// TIA Portal V16 export
// export: Created 2023-03-29T11:03:43.8543133Z, ExportSetting WithDefaults, DisplayName Totally Integrated Automation Portal, DisplayVersion V16 Update 6, DisplayName TIA Portal Version Control Interface, DisplayVersion V16 Update 2, DisplayName TIA Portal Openness, DisplayVersion V16 Update 6, DisplayName STEP 7 Professional, DisplayVersion V16 Update 6, DisplayName STEP 7 Safety, DisplayVersion V16, DisplayName WinCC Advanced, DisplayVersion V16 Update 6
VAR_GLOBAL   // PLC tag table "Default tag table"
   System_Byte AT %MB1 : Byte;
   FirstScan AT %M1.0 : Bool;
   DiagStatusUpdate AT %M1.1 : Bool;
   AlwaysTRUE AT %M1.2 : Bool;
   AlwaysFALSE AT %M1.3 : Bool;
   Clock_Byte AT %MB0 : Byte;
   Clock_10Hz AT %M0.0 : Bool;
   Clock_5Hz AT %M0.1 : Bool;
   "Clock_2.5Hz" AT %M0.2 : Bool;
   Clock_2Hz AT %M0.3 : Bool;
   "Clock_1.25Hz" AT %M0.4 : Bool;
   Clock_1Hz AT %M0.5 : Bool;
   "Clock_0.625Hz" AT %M0.6 : Bool;
   "Clock_0.5Hz" AT %M0.7 : Bool;
   trig_ustaw_czas AT %M206.1 : Bool;
   trig_pobierz_czas AT %M206.3 : Bool;
   "Bit_6-Wekt-Valve01_R" AT %M2000.6 : Bool;   // Bit-6 kasowanie alarmu
   "Bit_7-Wekt-Valve01_R" AT %M2000.7 : Bool;   // Bit trybu pracy napędu
   "Bit_5-Wekt-Valve01_R" AT %M2000.5 : Bool;   // Rozkaz zamykania
   "Bit_4-Wek_Valve01_R" AT %M2000.4 : Bool;   // Rozkaz otwieranie
   "Bit_0-Wekt_Valve01_R" AT %M2000.0 : Bool;   // Bit gotowośći / awarii
   "Bit_0-Wekt_Valve01_L" AT %M2001.0 : Bool;   // Bit Alarm/Gotowość (Alarm-=1, gotowość=0)
   "Bit_1-Wekt_Valve01_L" AT %M2001.1 : Bool;   // Bit potwierdzenia otwarcia
   "Bit_2-Wekt_Valve01_L" AT %M2001.2 : Bool;   // Bit wyboru trybu Zdalne=1 Remontowe=0
   "Bit_3-Wek_Valve01_L" AT %M2001.3 : Bool;   // Bit potwierdzenia zamknięcia
   "Bit_4-Wek_Valve01_L" AT %M2001.4 : Bool;   // Bit rozkazu na otwieranie
   "Bit_5-Wekt-Valve01_L" AT %M2001.5 : Bool;   // Bit rozkazu na zamykanie
   "Bit_6-Wekt-Valve01_L" AT %M2001.6 : Bool;   // Bit kasowania
   "Bit_7-Wekt-Valve01_L" AT %M2001.7 : Bool;   // Bit rodzaju sterowania aut =1 /manual= 0
   Byte_Wekt_Valve01_L AT %MB2001 : Byte;   // Lewy byte wektora napędu
   Byte_Wekt_Valve01_R AT %MB2000 : Byte;   // Prawy byte wektora napędu
   "I0.3" AT %I0.3 : Bool;
   "I0.4" AT %I0.4 : Bool;
   "I0.5" AT %I0.5 : Bool;
   "I0.6" AT %I0.6 : Bool;
   "Q0.3" AT %Q0.3 : Bool;
   "Q0.4" AT %Q0.4 : Bool;
   "Q0.5" AT %Q0.5 : Bool;
   "I6.4" AT %I6.4 : Bool;
   "I6.3" AT %I6.3 : Bool;
   "I6.2" AT %I6.2 : Bool;
   "I9.5" AT %I9.5 : Bool;
   "I9.6" AT %I9.6 : Bool;
   "I9.7" AT %I9.7 : Bool;
   "I3.1" AT %I3.1 : Bool;
   "I3.2" AT %I3.2 : Bool;
   "I3.3" AT %I3.3 : Bool;
   "I3.4" AT %I3.4 : Bool;
   "Q2.5" AT %Q2.5 : Bool;
   "Q2.6" AT %Q2.6 : Bool;
   "Q2.7" AT %Q2.7 : Bool;
   "I6.1" AT %I6.1 : Bool;
   "Bit_1-Wekt_Valve01_R" AT %M2000.1 : Bool;   // Bit potwierdzenia otwarcia
   "Byte_Wekt_POSITION_R(1)" AT %MB2002 : Byte;   // Prawy byte wektora napędu
   "Bit_0-Wekt_POSITION_R(1)" AT %M2002.0 : Bool;   // Bit gotowośći / awarii
   "Bit_1-Wekt_POSITION_R(1)" AT %M2002.1 : Bool;   // Bit potwierdzenia otwarcia
   "Bit_4-Wek_POSITION_R(1)" AT %M2002.4 : Bool;   // Rozkaz otwieranie
   "Bit_5-Wekt_POSITION_R(1)" AT %M2002.5 : Bool;   // Rozkaz zamykania
   "Bit_6-Wekt_POSITION_R(1)" AT %M2002.6 : Bool;   // Bit-6 kasowanie alarmu
   "Bit_7-Wekt_POSITION_R(1)" AT %M2002.7 : Bool;   // Bit trybu pracy napędu
   "Byte_Wekt_POSITION_L(1)" AT %MB2003 : Byte;   // Lewy byte wektora napędu
   "Bit_0-Wekt_POSITION_L(1)" AT %M2003.0 : Bool;   // Bit Alarm/Gotowość (Alarm-=1, gotowość=0)
   "Bit_1-Wekt_POSITION_L(1)" AT %M2003.1 : Bool;   // Bit potwierdzenia otwarcia
   "Bit_2-Wekt_POSITION_L(1)" AT %M2003.2 : Bool;   // Bit wyboru trybu Zdalne=1 Remontowe=0
   "Bit_3-Wek_POSITION_L(1)" AT %M2003.3 : Bool;   // Bit potwierdzenia zamknięcia
   "Bit_4-Wek_POSITION_L(1)" AT %M2003.4 : Bool;   // Bit rozkazu na otwieranie
   "Bit_5-Wekt_POSITION_L(1)" AT %M2003.5 : Bool;   // Bit rozkazu na zamykanie
   "Bit_6-Wekt_POSITION_L(1)" AT %M2003.6 : Bool;   // Bit kasowania
   "Bit_7-Wekt_POSITION_L(1)" AT %M2003.7 : Bool;   // Bit rodzaju sterowania aut =1 /manual= 0
   "Bit_2-Wekt_POSITION_R(1)" AT %M2002.2 : Bool;   // Bit wyboru trybu Zdalne=1 Remontowe=0
   "Bit_3-Wek_POSITION_R(1)" AT %M2002.3 : Bool;   // Bit potwierdzenia zamknięcia
   Tag_1 AT %M5000.0 : Bool;
   Tag_2 AT %M5000.1 : Bool;
   Tag_3 AT %M5000.3 : Bool;
   "I3.6" AT %I3.6 : Bool;
   "I3.7" AT %I3.7 : Bool;
   "I4.0" AT %I4.0 : Bool;
   "I3.5" AT %I3.5 : Bool;
   "I6.7" AT %I6.7 : Bool;
   "I6.6" AT %I6.6 : Bool;
   "I6.5" AT %I6.5 : Bool;
   "Q3.0" AT %Q3.0 : Bool;
   "Q3.1" AT %Q3.1 : Bool;
   "Q3.2" AT %Q3.2 : Bool;
   My_1Hz AT %M206.7 : Bool;
   "I1.1" AT %I1.1 : Bool;
   "I0.7" AT %I0.7 : Bool;
   "I1.0" AT %I1.0 : Bool;
   "I1.2" AT %I1.2 : Bool;
   "I7.0" AT %I7.0 : Bool;
   "I7.1" AT %I71.1 : Bool;
   "I7.2" AT %I7.2 : Bool;
   "Q3.4" AT %Q3.4 : Bool;
   "Q3.5" AT %Q3.5 : Bool;
   "Q3.6" AT %Q3.6 : Bool;
   "Q1.1" AT %Q1.1 : Bool;
   "Q2.0" AT %Q2.0 : Bool;
   "Q2.1" AT %Q2.1 : Bool;
   "I1.3" AT %I1.3 : Bool;
   "I1.4" AT %I1.4 : Bool;
   "I1.5" AT %I1.5 : Bool;
   "I2.0" AT %I2.0 : Bool;
   "I7.6" AT %I7.6 : Bool;
   "I7.7" AT %I7.7 : Bool;
   "I8.0" AT %I8.0 : Bool;
   "I7.3" AT %I7.3 : Bool;
   "I7.4" AT %I7.4 : Bool;
   "I7.5" AT %I7.5 : Bool;
   "I4.1" AT %I4.1 : Bool;
   "I4.2" AT %I4.2 : Bool;
   "I4.3" AT %I4.3 : Bool;
   "I4.4" AT %I4.4 : Bool;
   "I8.1" AT %I8.1 : Bool;
   "I8.2" AT %I8.2 : Bool;
   "I8.3" AT %I8.3 : Bool;
   "I4.5" AT %I4.5 : Bool;
   "I4.6" AT %I4.6 : Bool;
   "I4.7" AT %I4.7 : Bool;
   "I5.0" AT %I5.0 : Bool;
   "Q3.7" AT %Q3.7 : Bool;
   "Q4.0" AT %Q4.0 : Bool;
   "Q4.1" AT %Q4.1 : Bool;
   "Q2.2" AT %Q2.2 : Bool;
   "Q2.3" AT %Q2.3 : Bool;
   "Q2.4" AT %Q2.4 : Bool;
   "I2.1" AT %I2.1 : Bool;
   "I2.2" AT %I2.2 : Bool;
   "I2.3" AT %I2.3 : Bool;
   "I2.4" AT %I2.4 : Bool;
   "I8.4" AT %I8.4 : Bool;
   "I8.5" AT %I8.5 : Bool;
   "I8.6" AT %I8.6 : Bool;
   "I8.7" AT %I8.7 : Bool;
   "I9.0" AT %I9.0 : Bool;
   "I9.1" AT %I9.1 : Bool;
   "I5.1" AT %I5.1 : Bool;
   "I5.2" AT %I5.2 : Bool;
   "I5.3" AT %I5.3 : Bool;
   "I5.4" AT %I5.4 : Bool;
   "Q4.2" AT %Q4.2 : Bool;
   "Q4.3" AT %Q4.3 : Bool;
   "Q4.4" AT %Q4.4 : Bool;
   "I9.2" AT %I9.2 : Bool;
   "I9.3" AT %I9.3 : Bool;
   "I9.4" AT %I9.4 : Bool;
   "I0.0" AT %I0.0 : Bool;
   "I0.1" AT %I0.1 : Bool;
   "I0.2" AT %I0.2 : Bool;
   "Q0.6" AT %Q0.6 : Bool;
   "Q0.7" AT %Q0.7 : Bool;
   "Q1.0" AT %Q1.0 : Bool;
   "Q0.0" AT %Q0.0 : Bool;
   "Q0.1" AT %Q0.1 : Bool;
   "Q0.2" AT %Q0.2 : Bool;
   "I10.0" AT %I10.0 : Bool;
   setTime AT %M8.0 : Bool;   // ustaw zegar
   setData AT %M8.1 : Bool;   // ustaw datę
   isDaily AT %M80.7 : Bool;   // tryb sterowania dobowy
   isWeekiy AT %M81.0 : Bool;   // tryb sterowania tygodniowy
   isPowerOK AT %M81.2 : Bool;   // znacznik powrotu zasilania
   Tag_4 AT %Q6.7 : Bool;
   zbocze_dod_zegar AT %M47.0 : Bool;
   ResetErrorOB82 AT %M91.1 : Bool;
   "I5.5" AT %I5.5 : Bool;
   "I5.6" AT %I5.6 : Bool;
   "I5.7" AT %I5.7 : Bool;
   "I6.0" AT %I6.0 : Bool;
END_VAR
VAR_GLOBAL CONSTANT   // user constants
   analog_error_H : Word := 28538;
   CONST_BUFFER_OB82 : USInt := 200;
END_VAR
